// TwinCAT 3 PLC project IndraDriveTest
// ProgramVersion: 3.1.4023.0
// libraries:
//   Tc2_MC2, * (Beckhoff Automation GmbH)
//   Tc2_MC2_Drive, * (Beckhoff Automation GmbH)
//   Tc2_Standard, * (Beckhoff Automation GmbH)
//   Tc2_System, * (Beckhoff Automation GmbH)
//   Tc2_Utilities, * (Beckhoff Automation GmbH)
//   Tc3_Module, * (Beckhoff Automation GmbH)
// project tree:
//   AXIS CONTROL/ GVL_AXIS1.TcGVL (not stored), GVL_AXIS2.TcGVL (not stored), GVL_AXIS3.TcGVL (not stored), GVL_AXIS4.TcGVL (not stored), GVL_Safety_AXIS4.TcGVL (not stored), GVL_Safety_IO.TcGVL (not stored), P_AxisControl.TcPOU (not stored), ST_MC_CMD.TcDUT (not stored), ST_MC_ParametersAxis.TcDUT (not stored), ST_MC_Status.TcDUT (not stored)
//   INPUTS/Function Blocks/ FB_AnalogInputScaling.TcPOU (not stored), FB_JoystickInputScaling.TcPOU (not stored)
//   INPUTS/ G_Inputs.TcGVL (not stored), G_Sensors.TcGVL (not stored), P_Inputs.TcPOU
//   INPUTS/Struct/ ST_AnalogInput.TcDUT (not stored), ST_AnalogInputScaling.TcDUT, ST_AnalogInputStatus.TcDUT (not stored), ST_JoystickInputScaling.TcDUT
//   MACHINE CONTROL/ G_Parameters.TcGVL (not stored), G_Work.TcGVL, P_MachineControl.TcPOU
//   MACHINE CONTROL/InverseKinematics2d/ cosd_1.TcPOU (not stored), GVL_InverseKinematics.TcGVL, FB_InverseKin2d.TcPOU, rt_ceild_1.TcPOU, rt_floord_1.TcPOU (not stored), rt_remd_1.TcPOU (not stored)
//   MACHINE CONTROL/Struct/ ST_Parameters.TcDUT
//   OUTPUTS/ G_Outputs.TcGVL (not stored), P_Outputs.TcPOU
//   / PlcTask.TcTTO
//   POUs/ MAIN.TcPOU (not stored)
// real-time tasks:
//   TASK PlcTask: cycle T#10ms, priority 20, ADS port 350
// motion (NC):
//   TASK NC-Task 1 SAF: cycle T#2ms, priority 4, ADS port 501
//   TASK NC-Task 1 SVB: cycle T#10ms, priority 8, ADS port 511
//   AXIS Axis 1 - Bottom cylinder (id 1)
//     OtherSettings: AllowMotionCmdToSlave=true
//     encoder EncType=8
//       EncPara: MaxCount=#xffffffff
//         SoftEndMinControl: Enable=true, Range=21
//         SoftEndMaxControl: Enable=true, Range=290
//     drive DrvType=9
//       DrvPara: MaxCount=#xffffffff
//         Analog: VeloReferenz=100, VeloScale=6, TorqueSetpointScale=10, ScaleFactorActTorque=0.1
//         TimeComp: TaskDelayCycles=1
//     controller CtrType=1
//       CtrPara: PriorControlFactor=1
//         Observer: BandWidth=20
//   AXIS Axis 2 - Slew motor (id 2)
//     General: UnitName=Degree
//     Dynamic: AccelerationMaximum=55000, DecelerationMaximum=55000, Acceleration=30000, Deceleration=30000, Jerk=55000
//     Velo: SlowManual=200, FastManual=499, Maximum=6000
//     OtherSettings: AllowMotionCmdToSlave=true, PulseDistancePos=100, PulseDistanceNeg=100
//     encoder EncType=8
//       EncPara: MaxCount=#xffffffff
//         SoftEndMinControl: Enable=true, Range=-29000
//         SoftEndMaxControl: Enable=true, Range=29000
//     drive DrvType=9
//       DrvPara: MaxCount=#xffffffff, DriveControlDWord=#x00030000
//         Analog: VeloReferenz=5000, VeloScale=6, TorqueSetpointScale=10, ScaleFactorActTorque=0.1
//         TimeComp: TaskDelayCycles=1
//     controller CtrType=1
//       CtrPara: PriorControlFactor=1
//         Observer: BandWidth=20
//   AXIS Axis 3- Top cylinder (id 3)
//     OtherSettings: AllowMotionCmdToSlave=true
//     encoder EncType=8
//       EncPara: MaxCount=#xffffffff
//         SoftEndMinControl: Enable=true, Range=21
//         SoftEndMaxControl: Enable=true, Range=240
//     drive DrvType=9
//       DrvPara: MaxCount=#xffffffff
//         Analog: VeloScale=6, TorqueSetpointScale=10, ScaleFactorActTorque=0.1
//         TimeComp: TaskDelayCycles=1
//     controller CtrType=1
//       CtrPara: PriorControlFactor=1
//         Observer: BandWidth=20
//   AXIS Axis 4 - Winch motor (id 4)
//     OtherSettings: AllowMotionCmdToSlave=true
//     encoder EncType=19
//       EncPara: MaxCount=#xffffffff
//     drive DrvType=16
//       DrvPara: MaxCount=#xffffffff, DriveControlDWord=#x00000100
//         Analog: TorqueSetpointScale=10, ScaleFactorActTorque=0.1
//         TimeComp: TaskDelayCycles=1
//     controller CtrType=1
//       CtrPara: PriorControlFactor=1
//         Observer: BandWidth=20
//   AXIS Axis 5 (id 5)
//     OtherSettings: AllowMotionCmdToSlave=true
//     encoder EncType=8
//       EncPara: MaxCount=#x0036ee7f
//     drive DrvType=9
//       DrvPara: MaxCount=#xffffffff
//         Analog: VeloScale=6, TorqueSetpointScale=10, ScaleFactorActTorque=0.1
//         TimeComp: TaskDelayCycles=1
//     controller CtrType=1
//       CtrPara: PriorControlFactor=1
//         Observer: BandWidth=20
//   AXIS Axis 6 (id 6)
//     OtherSettings: AllowMotionCmdToSlave=true
//     encoder EncType=8
//       EncPara: MaxCount=#x0036ee7f
//     drive DrvType=9
//       DrvPara: MaxCount=#xffffffff
//         Analog: VeloScale=6, TorqueSetpointScale=10, ScaleFactorActTorque=0.1
//         TimeComp: TaskDelayCycles=1
//     controller CtrType=1
//       CtrPara: PriorControlFactor=1
//         Observer: BandWidth=20
//   AXIS Axis 7 (id 7)
//     OtherSettings: AllowMotionCmdToSlave=true
//     encoder EncType=8
//       EncPara: MaxCount=#x0036ee7f
//     drive DrvType=9
//       DrvPara: MaxCount=#xffffffff
//         Analog: VeloScale=6, TorqueSetpointScale=10, ScaleFactorActTorque=0.1
//         TimeComp: TaskDelayCycles=1
//     controller CtrType=1
//       CtrPara: PriorControlFactor=1
//         Observer: BandWidth=20
// I/O:
//   DEVICE Device 1 (EtherCAT), AmsNetId 5.107.189.26.2.1
//     Term 1 (EK1200) [EK1200-5000 EtherCAT Power supply (2A E-Bus)]
//       Term 2 (EL6910) [EL6910, TwinSAFE PLC]
//       Term 3 (EK1110) [EK1110 EtherCAT extension]
//     Term 4 (EK1818) [EK1818 EtherCAT IO-Coupler  (1A E-Bus, 8 Ch. Dig. In, 3ms, 4 Ch. Dig. Out 24V, 0,5A)]
//       Term 5 (EL3255) [EL3255 5Ch. potentiometer measurement with sensor supply]
//       Term 7 (EL9011) [EL9011 End Terminal]
//     Box 6 (AMI8000-0100) [AMI8000-0100 Servo motor 48 V DC, TwinSAFE]
//       modules: Module 1 (SAFETY)
//   DEVICE Device 5 (EtherCAT), AmsNetId 5.107.189.26.6.1
//     Drive 8 (IndraDrive MPB16/17) [IndraDrive MPB16/17]
//     Drive 9 (IndraDrive MPB20/21) [IndraDrive MPB20/21]
//     Drive 10 (IndraDrive MPB20/21) [IndraDrive MPB20/21]
// variable links:
//   NC-Task 1 SAF/Axes/Axis 5 <-> Device 5 (EtherCAT)/Drive 8 (IndraDrive MPB16/17)
//     Drive/Inputs/In/nDcOutputTime <-> InfoData/DcOutputShift
//     Drive/Inputs/In/nState1 <-> AT/Drive status word @bit 8
//     Drive/Inputs/In/nState2 <-> AT/Drive status word
//     Drive/Inputs/In/nState4 @bit 1 <-> WcState/InputToggle
//     Drive/Inputs/In/nState4 <-> WcState/WcState
//     Drive/Outputs/Out/nCtrl1 <-> MDT/Master control word @bit 8
//     Drive/Outputs/Out/nDataOut1 <-> MDT/Position command value
//     Enc/Inputs/In/nDataIn1 <-> AT/Position feedback value 1
//     Enc/Inputs/In/nDcInputTime <-> InfoData/DcInputShift
//     Enc/Inputs/In/nState4 @bit 1 <-> WcState/InputToggle
//     Enc/Inputs/In/nState4 <-> WcState/WcState
//   NC-Task 1 SAF/Axes/Axis 6 <-> Device 5 (EtherCAT)/Drive 9 (IndraDrive MPB20/21)
//     Drive/Inputs/In/nDcOutputTime <-> InfoData/DcOutputShift
//     Drive/Inputs/In/nState1 <-> AT/Drive status word @bit 8
//     Drive/Inputs/In/nState2 <-> AT/Drive status word
//     Drive/Inputs/In/nState4 @bit 1 <-> WcState/InputToggle
//     Drive/Inputs/In/nState4 <-> WcState/WcState
//     Drive/Outputs/Out/nCtrl1 <-> MDT/Master control word @bit 8
//     Drive/Outputs/Out/nDataOut1 <-> MDT/Position command value
//     Enc/Inputs/In/nDataIn1 <-> AT/Position feedback value 1
//     Enc/Inputs/In/nDcInputTime <-> InfoData/DcInputShift
//     Enc/Inputs/In/nState4 @bit 1 <-> WcState/InputToggle
//     Enc/Inputs/In/nState4 <-> WcState/WcState
//   NC-Task 1 SAF/Axes/Axis 7 <-> Device 5 (EtherCAT)/Drive 10 (IndraDrive MPB20/21)
//     Drive/Inputs/In/nDcOutputTime <-> InfoData/DcOutputShift
//     Drive/Inputs/In/nState1 <-> AT/Drive status word @bit 8
//     Drive/Inputs/In/nState2 <-> AT/Drive status word
//     Drive/Inputs/In/nState4 @bit 1 <-> WcState/InputToggle
//     Drive/Inputs/In/nState4 <-> WcState/WcState
//     Drive/Outputs/Out/nCtrl1 <-> MDT/Master control word @bit 8
//     Drive/Outputs/Out/nDataOut1 <-> MDT/Position command value
//     Enc/Inputs/In/nDataIn1 <-> AT/Position feedback value 1
//     Enc/Inputs/In/nDcInputTime <-> InfoData/DcInputShift
//     Enc/Inputs/In/nState4 @bit 1 <-> WcState/InputToggle
//     Enc/Inputs/In/nState4 <-> WcState/WcState
//   IndraDriveTest/IndraDriveTest Instance <-> Device 1 (EtherCAT)/Term 4 (EK1818)
//     PlcTask Inputs/G_Inputs.bAutoModeSelector <-> Channel 4/Input
//     PlcTask Inputs/G_Inputs.bGreenButton <-> Channel 6/Input
//     PlcTask Inputs/G_Inputs.bJoystickLeftEnable <-> Channel 7/Input
//     PlcTask Inputs/G_Inputs.bJoystickRightEnable <-> Channel 8/Input
//     PlcTask Inputs/G_Inputs.bManualModeSelector <-> Channel 3/Input
//     PlcTask Inputs/G_Inputs.bRedButton <-> Channel 5/Input
//     PlcTask Outputs/G_Outputs.bGreenButtonLight <-> Channel 9/Output
//     PlcTask Outputs/G_Outputs.bRedButtonLight <-> Channel 10/Output
//   IndraDriveTest/IndraDriveTest Instance <-> Device 1 (EtherCAT)/Term 4 (EK1818)/Term 5 (EL3255)
//     PlcTask Inputs/G_Inputs.stJoyLX.nValue <-> AI Standard Channel 1/Value
//     PlcTask Inputs/G_Inputs.stJoyLX.stStatus <-> AI Standard Channel 1/Status
//     PlcTask Inputs/G_Inputs.stJoyLY.nValue <-> AI Standard Channel 2/Value
//     PlcTask Inputs/G_Inputs.stJoyLY.stStatus <-> AI Standard Channel 2/Status
//     PlcTask Inputs/G_Inputs.stJoyRX.nValue <-> AI Standard Channel 3/Value
//     PlcTask Inputs/G_Inputs.stJoyRX.stStatus <-> AI Standard Channel 3/Status
//     PlcTask Inputs/G_Inputs.stJoyRY.nValue <-> AI Standard Channel 4/Value
//     PlcTask Inputs/G_Inputs.stJoyRY.stStatus <-> AI Standard Channel 4/Status
//   IndraDriveTest/IndraDriveTest Instance <-> NC-Task 1 SAF/Axes/Axis 1 - Bottom cylinder
//     PlcTask Inputs/GVL_AXIS1.BCAxis.NcToPlc <-> Outputs/ToPlc
//     PlcTask Outputs/GVL_AXIS1.BCAxis.PlcToNc <-> Inputs/FromPlc
//   IndraDriveTest/IndraDriveTest Instance <-> NC-Task 1 SAF/Axes/Axis 2 - Slew motor
//     PlcTask Inputs/GVL_AXIS2.SJAxis.NcToPlc <-> Outputs/ToPlc
//     PlcTask Outputs/GVL_AXIS2.SJAxis.PlcToNc <-> Inputs/FromPlc
//   IndraDriveTest/IndraDriveTest Instance <-> NC-Task 1 SAF/Axes/Axis 3- Top cylinder
//     PlcTask Inputs/GVL_AXIS3.TCAxis.NcToPlc <-> Outputs/ToPlc
//     PlcTask Outputs/GVL_AXIS3.TCAxis.PlcToNc <-> Inputs/FromPlc

CONFIGURATION IndraDriveTest
    RESOURCE PLC ON TwinCAT3
        TASK PlcTask(INTERVAL := T#10ms, PRIORITY := 20);
        PROGRAM MAIN WITH PlcTask : MAIN;
    END_RESOURCE
END_CONFIGURATION

// ---- INPUTS/Struct/ST_AnalogInputScaling.TcDUT
TYPE ST_AnalogInputScaling :
STRUCT
	fMaxInputValue 			: LREAL;	// tunable max input value 
	fMinInputValue			: LREAL;	// tunable min input value  
	fMaxOutputValue  		: LREAL;	// max sensor output value
	fMinOutputValue  		: LREAL;	// min sensor output value	
END_STRUCT
END_TYPE

// ---- INPUTS/Struct/ST_JoystickInputScaling.TcDUT
TYPE ST_JoystickInputScaling :
STRUCT
	fMaxInputValue			: LREAL;	// tunable max input value
	fMinInputValue 			: LREAL;	// tunable min input value
	fNeutralInputValue  	: LREAL;	// tunable neutral input value
	fNeutralDeadband		: LREAL;	// tunable dead_band value
	fMaxOutputValue  		: LREAL;	// normalized max output value
	fMinOutputValue  		: LREAL;	// normalized min output value
	fNeutralOutputValue  	: LREAL;	// normalized neutral output value
END_STRUCT
END_TYPE

// ---- MACHINE CONTROL/Struct/ST_Parameters.TcDUT
TYPE ST_Parameters :
STRUCT
	fCyclicTime 					: LREAL := 0.001; // [s]
	
	stJoystickInputScalingLeftX 		: ST_JoystickInputScaling := (fMaxInputValue := 20482.0, fMinInputValue := 11828.0, fNeutralInputValue := 16267, fNeutralDeadband := 100.0, fMaxOutputValue := 1.0, fMinOutputValue := -1.0, fNeutralOutputValue := 0.0);
	stJoystickInputScalingLeftY 		: ST_JoystickInputScaling := (fMaxInputValue := 20720.0, fMinInputValue := 11950.0, fNeutralInputValue := 16475, fNeutralDeadband := 100.0, fMaxOutputValue := 1.0, fMinOutputValue := -1.0, fNeutralOutputValue := 0.0);
	stJoystickInputScalingRightX 		: ST_JoystickInputScaling := (fMaxInputValue := 20550.0, fMinInputValue := 11800.0, fNeutralInputValue := 16297, fNeutralDeadband := 100.0, fMaxOutputValue := 1.0, fMinOutputValue := -1.0, fNeutralOutputValue := 0.0);
	stJoystickInputScalingRightY 		: ST_JoystickInputScaling := (fMaxInputValue := 20500.0, fMinInputValue := 11800.0, fNeutralInputValue := 16225, fNeutralDeadband := 100.0, fMaxOutputValue := 1.0, fMinOutputValue := -1.0, fNeutralOutputValue := 0.0);

		
END_STRUCT
END_TYPE

// ---- MACHINE CONTROL/G_Work.TcGVL
{attribute 'qualified_only'}
VAR_GLOBAL
	bManualMode 			: BOOL;
	bAutoMode 				: BOOL;
	bWinchEnable 			: BOOL;
	bCylEnable 				: BOOL;
	fWinchControlInput 		: LREAL;
	fWinchTime				: LREAL;
	fCylControlInput 		: LREAL;
	fCylTime				: LREAL;
	fVelRefWinch 			: LREAL;
	fPosRefWinch 			: LREAL;
	fControlSignWinch		: LREAL;
	fVelRefCyl 				: LREAL;
	fPosRefCyl 				: LREAL;
	fControlSignCyl			: LREAL;
	fPositionErrorWinch_mm 	: LREAL;
	fPositionErrorCylinder_mm : LREAL;
END_VAR

// ---- MACHINE CONTROL/InverseKinematics2d/GVL_InverseKinematics.TcGVL
{attribute 'qualified_only'}
VAR_GLOBAL
	fTooltipXCoordGlobalIni: LREAL := 2.8;
	fTooltipYCoordGlobalIni: LREAL := 0.0;
	//fTooltipZCoordGlobalIni: LREAL := 0.0;
	fAngleMainArmInverse :	LREAL;
	fAngleKnuckleArmInverse : LREAL;
	fStrokeActuatorMainInverse : LREAL;
	fStrokeActuatorKnuckleInverse : LREAL;
END_VAR

// ---- INPUTS/P_Inputs.TcPOU
PROGRAM P_Inputs
VAR
	fbJoystickLeftVert 					: FB_JoystickInputScaling;
	fbJoystickLeftHor 					: FB_JoystickInputScaling;
	
	fbJoystickRightVert 				: FB_JoystickInputScaling;
	fbJoystickRightHor 					: FB_JoystickInputScaling;
	
	
END_VAR

 fbJoystickLeftVert(
	bEnable := G_Work.bManualMode,
	nRawInput := G_Inputs.stJoyLY.nValue,
	stJoystickInputScaling := G_Parameters.stParam.stJoystickInputScalingLeftY,
	fNormalizedOutput => G_Sensors.fJoystickLeftNormalizedY
);

fbJoystickLeftHor(
	bEnable := G_Work.bManualMode,
	nRawInput := G_Inputs.stJoyLX.nValue,
	stJoystickInputScaling := G_Parameters.stParam.stJoystickInputScalingLeftX,
	fNormalizedOutput => G_Sensors.fJoystickLeftNormalizedX
);

IF G_Sensors.fJoystickLeftNormalizedX < 0 THEN
	G_Sensors.MCDirectionAxis1 := MC_Positive_Direction;
ELSIF G_Sensors.fJoystickLeftNormalizedX > 0 THEN
	G_Sensors.MCDirectionAxis1 := MC_Negative_Direction;	
//ELSE
//	G_Sensors.MCDirectionAxis1 := MC_Current_Direction;
END_IF


fbJoystickRightVert(
	bEnable := G_Work.bManualMode,
	nRawInput := G_Inputs.stJoyRY.nValue,
	stJoystickInputScaling := G_Parameters.stParam.stJoystickInputScalingRightY,
	fNormalizedOutput => G_Sensors.fJoystickRightNormalizedY
);

fbJoystickRightHor(
	bEnable := G_Work.bManualMode,
	nRawInput := G_Inputs.stJoyRX.nValue,
	stJoystickInputScaling := G_Parameters.stParam.stJoystickInputScalingRightX,
	fNormalizedOutput => G_Sensors.fJoystickRightNormalizedX
);

END_PROGRAM

// ---- MACHINE CONTROL/InverseKinematics2d/FB_InverseKin2d.TcPOU
FUNCTION_BLOCK FB_InverseKin2d
VAR_INPUT
	fPtXd: LREAL;
	fPtYd: LREAL;
	fTheta1: LREAL;
END_VAR
VAR_OUTPUT
	fStrokeActuatorMain: LREAL;
	fStrokeActuatorKnuckle: LREAL;
	fTheta3: LREAL;
	fTheta4: LREAL;
END_VAR
VAR
	h: LREAL;
	ThetaB: LREAL;
	ThetaB_tmp: LREAL;
	b_a_tmp: LREAL;
	a_tmp: LREAL;
	i0_cosd: cosd;
END_VAR


(* MATLAB Function: '<Root>/Inverse kinematics function' *)
(* clc; close all; clear; *)
(* MATLAB Function 'Inverse kinematics function': '<S1>:1' *)
(* Inputs *)
(* Desired global coordinates *)
(* fPtXd		= 0.75 + 1.5; *)
(* fPtYd		= 1.065 + 0.176; *)

(* %     fPtXd		= 0.75 + 0.716; *)
(* %  	fPtYd		= 1.065 + 0.705; *)
(* Platform constants *)
(* '<S1>:1:14' h0 = 1.0; *)
(* '<S1>:1:15' l0 = 0.75; *)
(* Crane constants *)
(* '<S1>:1:18' h1 = 1.334 + 0.065; *)
(* '<S1>:1:19' lm = 1.5; *)
(* '<S1>:1:20' lk = 1.158; *)
(* Calculate position of a2 as function of Theta1 *)
(* '<S1>:1:23' a2x = l0*cos(fTheta1) + h1*cos(fTheta1 + pi/2); *)
(* '<S1>:1:24' a2y = h0 + l0*sin(fTheta1) + h1*sin(fTheta1 + pi/2); *)
(* '<S1>:1:26' h = sqrt((fPtXd - a2x)^2 + (fPtYd - a2y)^2); *)
a_tmp := fPtXd - ((COS(fTheta1 + 1.5707963267948966) * 1.399) + (0.75 * COS(fTheta1)));
b_a_tmp := fPtYd - (((0.75 * SIN(fTheta1)) + 1.0) + (SIN(fTheta1 + 1.5707963267948966) * 1.399));
h := SQRT((a_tmp * a_tmp) + (b_a_tmp * b_a_tmp));
(* '<S1>:1:27' phi = atan((fPtYd - a2y) / (fPtXd - a2x)); *)
(* Calculate ThetaA and ThetaB *)
(* '<S1>:1:30' ThetaA = acos ((lm^2 + h^2 - lk^2) / (2*lm*h)); *)
(* '<S1>:1:31' ThetaB = acos ((lk^2 + lm^2 - h^2) / (2*lm*lk)); *)
ThetaB_tmp := h * h;
ThetaB := ACOS((3.5909639999999996 - ThetaB_tmp) / 3.4739999999999998);
(* '<S1>:1:33' fTheta3 = ThetaA + phi - fTheta1; *)
fTheta3 := (ACOS(((ThetaB_tmp + 2.25) - 1.3409639999999998) / (3.0 * h)) + ATAN(b_a_tmp / a_tmp)) - fTheta1;
(* '<S1>:1:34' fTheta4 = ThetaB - pi/2; *)
(* '<S1>:1:36' fTheta3deg = rad2deg(fTheta3); *)
(* '<S1>:1:37' fTheta4deg = rad2deg(fTheta4); *)
(* Crane constant parameters *)
(* '<S1>:1:40' fLengthP2PMainArm			= lm; *)
(* '<S1>:1:41' fLengthP2PKnuckleArm		= lk; *)
(* '<S1>:1:43' fLengthAMain				= 0.614; *)
(* '<S1>:1:44' fLengthBMain				= 0.571; *)
(* '<S1>:1:45' fMinLengthActuatorMain		= 0.692; *)
(* '<S1>:1:46' fMaxStrokeActuatorMain		= 0.320; *)
(* '<S1>:1:48' fOffsetAngleDegMainAct		= 62.1; *)
(* '<S1>:1:50' fLengthAKnuckle				= 0.767; *)
(* '<S1>:1:51' fLengthBKnuckle				= 0.184; *)
(* '<S1>:1:52' fMinLengthActuatorKnuckle	= 0.627; *)
(* '<S1>:1:53' fMaxStrokeActuatorKnuckle	= 0.260; *)
(* '<S1>:1:55' fOffsetAngleDegKnuckleAct	= 86.3; *)
(* '<S1>:1:58' fAngleMainArmAct			= fTheta3deg + fOffsetAngleDegMainAct; *)
(* '<S1>:1:59' fAngleKnuckleArmAct         = fTheta4deg + fOffsetAngleDegKnuckleAct; *)
(* '<S1>:1:61' fLengthActuatorMain         = sqrt(fLengthAMain^2 + fLengthBMain^2 -(2*fLengthAMain*fLengthBMain*cosd(fAngleMainArmAct))); *)
(* '<S1>:1:62' fStrokeActuatorMain         = fLengthActuatorMain - fMinLengthActuatorMain; *)
a_tmp := (57.295779513082323 * fTheta3) + 62.1;
b_a_tmp := a_tmp;
i0_cosd(x := b_a_tmp);
(* Outport: '<Root>/fStrokeActuatorMain' incorporates:
 *  MATLAB Function: '<Root>/Inverse kinematics function' *)
fStrokeActuatorMain := SQRT(0.70303699999999991 - (0.70118799999999992 * b_a_tmp)) - 0.692;
(* MATLAB Function: '<Root>/Inverse kinematics function' *)
(* '<S1>:1:64' if fStrokeActuatorMain < 0 *)
b_a_tmp := a_tmp;
i0_cosd(x := b_a_tmp);

IF (SQRT(0.70303699999999991 - (0.70118799999999992 * b_a_tmp)) - 0.692) < 0.0 THEN 
    (* Outport: '<Root>/fStrokeActuatorMain' *)
    (* '<S1>:1:65' fStrokeActuatorMain = 0; *)
    fStrokeActuatorMain := 0.0;
END_IF;

(* '<S1>:1:70' fLengthActuatorKnuckle         = sqrt(fLengthAKnuckle^2 + fLengthBKnuckle^2 -(2*fLengthAKnuckle*fLengthBKnuckle*cosd(fAngleKnuckleArmAct))); *)
(* '<S1>:1:71' fStrokeActuatorKnuckle         = fLengthActuatorKnuckle - fMinLengthActuatorKnuckle; *)
a_tmp := ((ThetaB - 1.5707963267948966) * 57.295779513082323) + 86.3;
b_a_tmp := a_tmp;
i0_cosd(x := b_a_tmp);
(* Outport: '<Root>/fStrokeActuatorKnuckle' incorporates:
 *  MATLAB Function: '<Root>/Inverse kinematics function' *)
fStrokeActuatorKnuckle := SQRT(0.62214500000000006 - (0.282256 * b_a_tmp)) - 0.627;
(* MATLAB Function: '<Root>/Inverse kinematics function' *)
(* '<S1>:1:73' if fStrokeActuatorKnuckle < 0 *)
b_a_tmp := a_tmp;
i0_cosd(x := b_a_tmp);

IF (SQRT(0.62214500000000006 - (0.282256 * b_a_tmp)) - 0.627) < 0.0 THEN 
    (* Outport: '<Root>/fStrokeActuatorKnuckle' *)
    (* '<S1>:1:74' fStrokeActuatorKnuckle = 0; *)
    fStrokeActuatorKnuckle := 0.0;
END_IF;

(* Outport: '<Root>/fTheta4' incorporates:
 *  MATLAB Function: '<Root>/Inverse kinematics function' *)
fTheta4 := ThetaB - 1.5707963267948966;

END_FUNCTION_BLOCK

// ---- MACHINE CONTROL/InverseKinematics2d/rt_ceild_1.TcPOU
FUNCTION rt_ceild_1 : LREAL
VAR_INPUT
	u: LREAL;
END_VAR
VAR
END_VAR


rt_ceild := DINT_TO_LREAL(TRUNC(u));

IF u = rt_ceild THEN 
    rt_ceild := u;
ELSIF u >= 0.0 THEN 
    rt_ceild := rt_ceild + 1.0;
END_IF;

END_FUNCTION

// ---- MACHINE CONTROL/P_MachineControl.TcPOU
PROGRAM P_MachineControl
VAR
	fbInverse					: FB_InverseKin2d;
END_VAR

G_Work.bManualMode := G_Inputs.bManualModeSelector;
G_Work.bAutoMode := G_Inputs.bAutoModeSelector;

fbInverse(
	fPtXd := GVL_InverseKinematics.fTooltipXCoordGlobalIni, 
	fPtYd := GVL_InverseKinematics.fTooltipYCoordGlobalIni, 
	fTheta1: LREAL := 0;
	
	fTheta3 => GVL_InverseKinematics.fAngleMainArmInverse, 
	fTheta4 => GVL_InverseKinematics.fAngleKnuckleArmInverse,
	fStrokeActuatorMain => GVL_InverseKinematics.fStrokeActuatorMainInverse,
	fStrokeActuatorKnuckle => GVL_InverseKinematics.fStrokeActuatorKnuckleInverse,	
);

END_PROGRAM

// ---- OUTPUTS/P_Outputs.TcPOU
PROGRAM P_Outputs
VAR
END_VAR

///////////////////// Lights //////////////////////////////

IF G_Inputs.bRedButton THEN 
	G_Outputs.bRedButtonLight := FALSE;
ELSE 
	G_Outputs.bRedButtonLight := TRUE;
END_IF

IF G_Inputs.bGreenButton THEN 
	G_Outputs.bGreenButtonLight := TRUE;
ELSE 
	G_Outputs.bGreenButtonLight := FALSE;
END_IF


IF G_Inputs.bManualModeSelector OR G_Inputs.bAutoModeSelector THEN
	G_Outputs.bGreenButtonLight := FALSE;
	G_Outputs.bRedButtonLight := TRUE;
ELSE
	G_Outputs.bGreenButtonLight := TRUE;
	G_Outputs.bRedButtonLight := FALSE;
END_IF

END_PROGRAM
